// TIA Portal project "TrainingModules2" (V15.1)

(* hardware
DEVICE "S71500/ET200MP station_1"  S7-1500 station
   slot 0: "Rail_0"  Rack  6ES7 590-1***0-0AA0
   slot 1: "PLC_1"  CPU 1516-3 PN/DP  6ES7 516-3AN01-0AB0  V2.6
      slot 3: "CPU display_1"  6ES7591-1BA00-0AA0
*)

// ===== PLC "PLC_1"  CPU 1516-3 PN/DP =====

VAR_GLOBAL   // PLC tag table "Control Panel"
   "Auto Mode" AT %I0.0 : Bool;   // Automaitc Mode Switch
   "Auto Mode Start PB" AT %I0.1 : Bool;   // Auto Mode Start Push Button
   "Auto Mode Stop PB" AT %I0.2 : Bool;   // Auto Mode Stop Push Button
   "Manual Mode" AT %I0.3 : Bool;   // Manual Mode Switch
   "Reset Counter" AT %I0.4 : Bool;   // Reset Part Counter
   "EStop" AT %I0.5 : Bool;   // Emergency Stop
   "Start Light" AT %Q0.0 : Bool;   // Start Push Button Light
   "Stop Light" AT %Q0.1 : Bool;   // Stop Push Button Light
   "Reset Light" AT %Q0.2 : Bool;   // Reset Push Button Light
   "Part Entry Counter" AT %QD100 : DInt;   // Part Entry Counter
   "Garbage" AT %M10.0 : Bool;   // Storage for Last Cycle, Not Used
   "Garbage2" AT %M10.1 : Bool;   // Storage for Last Cycle, Not Used
END_VAR

VAR_GLOBAL   // PLC tag table "Conveyor"
   "Tall Sensor" AT %I0.6 : Bool;   // Second Level Height Sensor
   "Short Sensor" AT %I0.7 : Bool;   // First Level Height Sensor
   "Conveyor_Loader_Entry" AT %I1.2 : Bool;   // Entering the Main Conveyor
   "Conveyor_Left_Entry" AT %I1.3 : Bool;   // Left Conveyor Entry Sensor
   "Conveyor_Right_Entry" AT %I1.4 : Bool;   // Right Conveyor Entry Sensor
   "Conveyor_Turntable_Entry" AT %I1.5 : Bool;   // Entering the Turntable
   "Feeder Conveyor" AT %Q0.3 : Bool;   // Feeder Conveyor Actuator
   "Entry Conveyor" AT %Q0.4 : Bool;   // Entry Conveyor Actuator
   "Left Conveyor" AT %Q1.0 : Bool;   // Left Conveyor Actuator
   "Right Conveyor" AT %Q1.1 : Bool;   // Right Conveyor Actuator
   "Green Indicator" AT %Q1.2 : Bool;   // Green Light Indicator
   "Yellow Indicator" AT %Q1.3 : Bool;   // Yellow Light Indicator
   "Red Indicator" AT %Q1.4 : Bool;   // Red Light Indicator
   "Emitter" AT %Q1.5 : Bool;   // Send Parts
   "Remover Left" AT %Q1.6 : Bool;   // Remove Parts Left Side
   "Remover Right" AT %Q1.7 : Bool;   // Remove Parts Right SIde
END_VAR

VAR_GLOBAL   // PLC tag table "Turntable"
   "TT_Front" AT %I1.0 : Bool;   // Turn Table Entry Sensor
   "TT_Back" AT %I1.1 : Bool;   // Turn Table Exit Sensor
   "Home" AT %I1.6 : Bool;   // Turn Table Homed
   "Rotated" AT %I1.7 : Bool;   // Turn Table Rotated
   "Load (Right)" AT %Q0.5 : Bool;   // Load Right Conveyor (TT)
   "Unload (Left)" AT %Q0.6 : Bool;   // Load Left Conveyor (TT)
   "Turn CC" AT %Q0.7 : Bool;   // Turn Table Rotate Counter CLockwise
END_VAR

VAR_GLOBAL   // PLC tag table "Part Buffer"
   "Part_Space_5" AT %MW0 : Int;   // Part Buffer 5
   "Part_Space_4" AT %MW2 : Int;   // Part Buffer 4
   "Part_Space_3" AT %MW4 : Int;   // Part Buffer 3
   "Part_Space_2" AT %MW6 : Int;   // Part Buffer 2
   "Part_Space_1" AT %MW8 : Int;   // Part Buffer 1
END_VAR

DATA_BLOCK "Data_Organization"   // DB1
{ S7_Optimized_Access := 'TRUE' }
VERSION : 0.1
// stored: InstanceOfName Controller
"Controller"
BEGIN
END_DATA_BLOCK

FUNCTION_BLOCK "Controller"   // FB1, LAD
{ S7_Optimized_Access := 'TRUE' }
VERSION : 0.1
   VAR
      "Conveyor Logic_Feeder" : "Conveyor Logic";
      "Turntable Logic" : "Turntable Logic";
      "Conveyor Logic_Entry" : "Conveyor Logic";
      "Conveyor Logic_Left" : "Conveyor Logic";
      "Conveyor Logic_Right" : "Conveyor Logic";
   END_VAR
   VAR_TEMP   // added for the SCL form of the ladder/FBD networks
      _w1 : Bool;
   END_VAR
BEGIN

REGION Network 1: Call the Send and Receive function
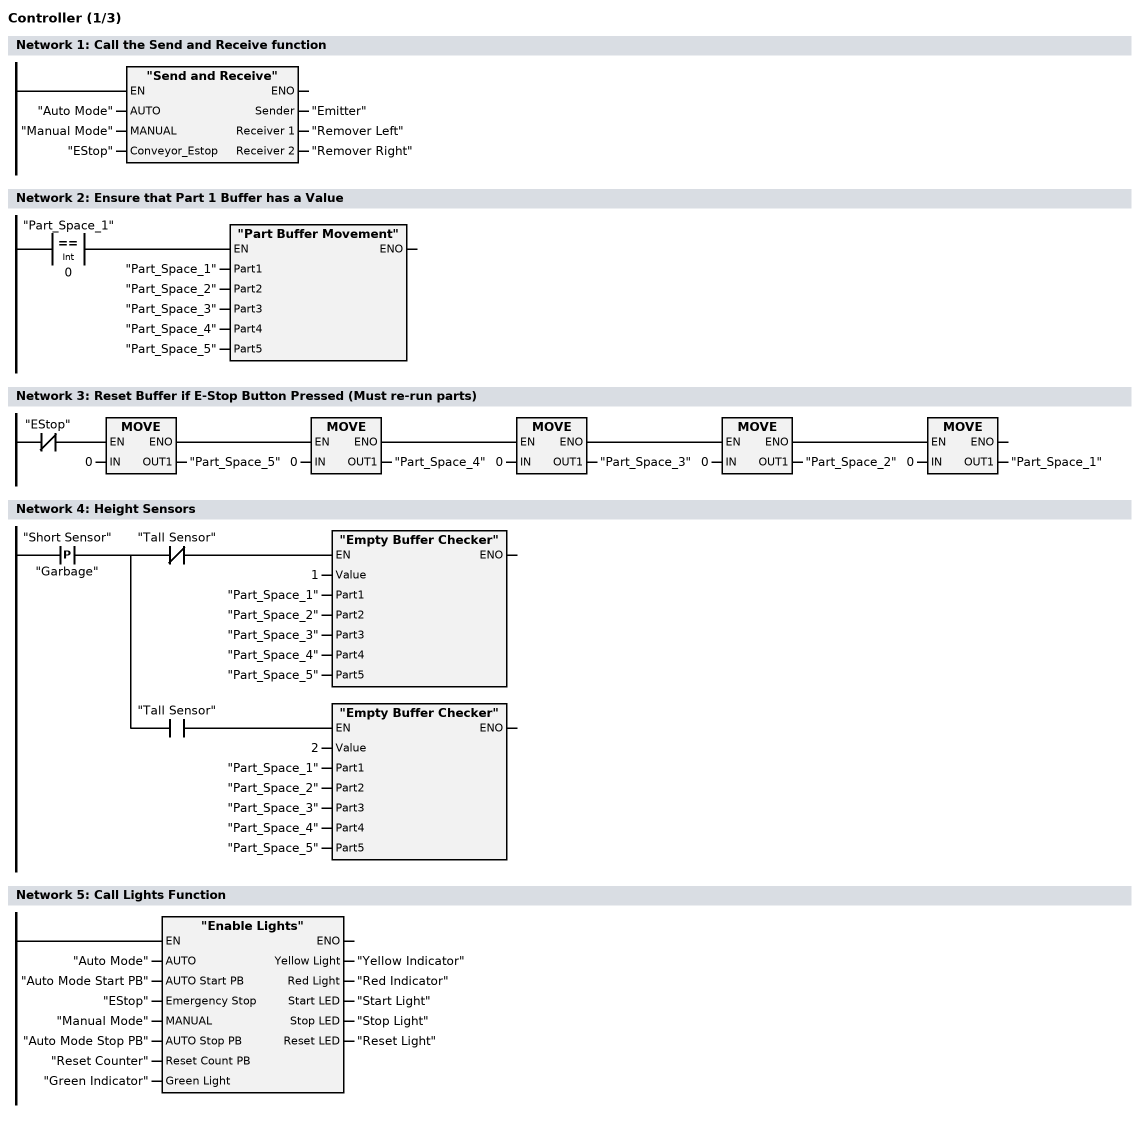
   RUNG wire#powerrail
      "Send and Receive"(AUTO := "Auto Mode", MANUAL := "Manual Mode", Conveyor_Estop := "EStop", Sender => "Emitter", "Receiver 1" => "Remover Left", "Receiver 2" => "Remover Right")
   END_RUNG
   // the same network as SCL:
   "Send and Receive"(AUTO := "Auto Mode",
                      MANUAL := "Manual Mode",
                      Conveyor_Estop := "EStop",
                      Sender => "Emitter",
                      "Receiver 1" => "Remover Left",
                      "Receiver 2" => "Remover Right");
END_REGION

REGION Network 2: Ensure that Part 1 Buffer has a Value
   RUNG wire#powerrail
      { S7_Templates := "SrcType := Int" } EQ_Contact(in1 := "Part_Space_1", in2 := 0)
      "Part Buffer Movement"(Part1 := "Part_Space_1", Part2 := "Part_Space_2", Part3 := "Part_Space_3", Part4 := "Part_Space_4", Part5 := "Part_Space_5")
   END_RUNG
   // the same network as SCL:
   IF "Part_Space_1" = 0 THEN
       "Part Buffer Movement"(Part1 := "Part_Space_1",
                              Part2 := "Part_Space_2",
                              Part3 := "Part_Space_3",
                              Part4 := "Part_Space_4",
                              Part5 := "Part_Space_5");
   END_IF;
END_REGION

REGION Network 3: Reset Buffer if E-Stop Button Pressed (Must re-run parts)
   RUNG wire#powerrail
      I_Contact( "EStop" )
      Move(in := 0, out1 => "Part_Space_5")
      Move(in := 0, out1 => "Part_Space_4")
      Move(in := 0, out1 => "Part_Space_3")
      Move(in := 0, out1 => "Part_Space_2")
      Move(in := 0, out1 => "Part_Space_1")
   END_RUNG
   // the same network as SCL:
   IF NOT "EStop" THEN
       "Part_Space_5" := 0;
       "Part_Space_4" := 0;
       "Part_Space_3" := 0;
       "Part_Space_2" := 0;
       "Part_Space_1" := 0;
   END_IF;
END_REGION

REGION Network 4: Height Sensors
   RUNG wire#powerrail
      P_Contact(operand := "Short Sensor", bit := "Garbage")
      wire#w1
      I_Contact( "Tall Sensor" )
      "Empty Buffer Checker"(Value := 1, Part1 := "Part_Space_1", Part2 := "Part_Space_2", Part3 := "Part_Space_3", Part4 := "Part_Space_4", Part5 := "Part_Space_5")
   END_RUNG
   RUNG wire#w1
      Contact( "Tall Sensor" )
      "Empty Buffer Checker"(Value := 2, Part1 := "Part_Space_1", Part2 := "Part_Space_2", Part3 := "Part_Space_3", Part4 := "Part_Space_4", Part5 := "Part_Space_5")
   END_RUNG
   // the same network as SCL:
   #_w1 := "Short Sensor" AND NOT "Garbage";   // rising edge of "Short Sensor"
   "Garbage" := "Short Sensor";
   IF #_w1 AND NOT "Tall Sensor" THEN
       "Empty Buffer Checker"(Value := 1,
                              Part1 := "Part_Space_1",
                              Part2 := "Part_Space_2",
                              Part3 := "Part_Space_3",
                              Part4 := "Part_Space_4",
                              Part5 := "Part_Space_5");
   END_IF;
   IF #_w1 AND "Tall Sensor" THEN
       "Empty Buffer Checker"(Value := 2,
                              Part1 := "Part_Space_1",
                              Part2 := "Part_Space_2",
                              Part3 := "Part_Space_3",
                              Part4 := "Part_Space_4",
                              Part5 := "Part_Space_5");
   END_IF;
END_REGION

REGION Network 5: Call Lights Function
   RUNG wire#powerrail
      "Enable Lights"(AUTO := "Auto Mode", "AUTO Start PB" := "Auto Mode Start PB", "Emergency Stop" := "EStop", MANUAL := "Manual Mode", "AUTO Stop PB" := "Auto Mode Stop PB", "Reset Count PB" := "Reset Counter", "Green Light" := "Green Indicator", "Yellow Light" => "Yellow Indicator", "Red Light" => "Red Indicator", "Start LED" => "Start Light", "Stop LED" => "Stop Light", "Reset LED" => "Reset Light")
   END_RUNG
   // the same network as SCL:
   "Enable Lights"(AUTO := "Auto Mode",
                   "AUTO Start PB" := "Auto Mode Start PB",
                   "Emergency Stop" := "EStop",
                   MANUAL := "Manual Mode",
                   "AUTO Stop PB" := "Auto Mode Stop PB",
                   "Reset Count PB" := "Reset Counter",
                   "Green Light" := "Green Indicator",
                   "Yellow Light" => "Yellow Indicator",
                   "Red Light" => "Red Indicator",
                   "Start LED" => "Start Light",
                   "Stop LED" => "Stop Light",
                   "Reset LED" => "Reset Light");
END_REGION

REGION Network 6: Call Feeder Conveyor Logic
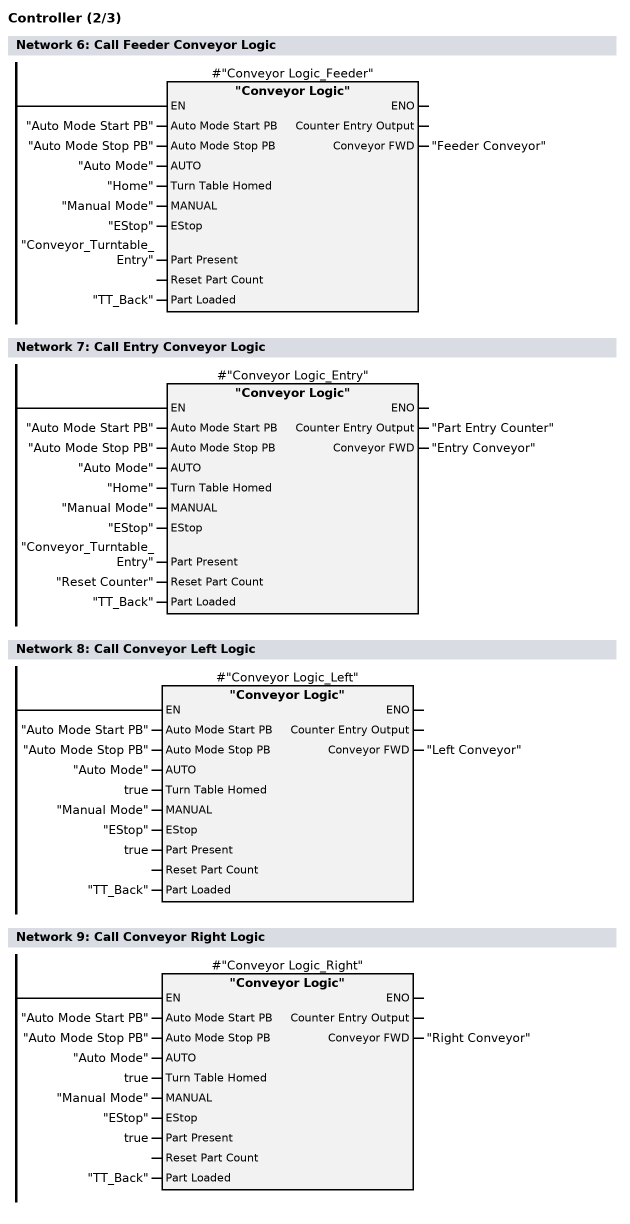
   RUNG wire#powerrail
      #"Conveyor Logic_Feeder"("Auto Mode Start PB" := "Auto Mode Start PB", "Auto Mode Stop PB" := "Auto Mode Stop PB", AUTO := "Auto Mode", "Turn Table Homed" := "Home", MANUAL := "Manual Mode", EStop := "EStop", "Part Present" := "Conveyor_Turntable_Entry", "Reset Part Count" :=, "Part Loaded" := "TT_Back", "Counter Entry Output" =>, "Conveyor FWD" => "Feeder Conveyor")
   END_RUNG
   // the same network as SCL:
   #"Conveyor Logic_Feeder"("Auto Mode Start PB" := "Auto Mode Start PB",   // "Conveyor Logic"
                           "Auto Mode Stop PB" := "Auto Mode Stop PB",
                           AUTO := "Auto Mode",
                           "Turn Table Homed" := "Home",
                           MANUAL := "Manual Mode",
                           EStop := "EStop",
                           "Part Present" := "Conveyor_Turntable_Entry",
                           "Part Loaded" := "TT_Back",
                           "Conveyor FWD" => "Feeder Conveyor");
END_REGION

REGION Network 7: Call Entry Conveyor Logic
   RUNG wire#powerrail
      #"Conveyor Logic_Entry"("Auto Mode Start PB" := "Auto Mode Start PB", "Auto Mode Stop PB" := "Auto Mode Stop PB", AUTO := "Auto Mode", "Turn Table Homed" := "Home", MANUAL := "Manual Mode", EStop := "EStop", "Part Present" := "Conveyor_Turntable_Entry", "Reset Part Count" := "Reset Counter", "Part Loaded" := "TT_Back", "Counter Entry Output" => "Part Entry Counter", "Conveyor FWD" => "Entry Conveyor")
   END_RUNG
   // the same network as SCL:
   #"Conveyor Logic_Entry"("Auto Mode Start PB" := "Auto Mode Start PB",   // "Conveyor Logic"
                           "Auto Mode Stop PB" := "Auto Mode Stop PB",
                           AUTO := "Auto Mode",
                           "Turn Table Homed" := "Home",
                           MANUAL := "Manual Mode",
                           EStop := "EStop",
                           "Part Present" := "Conveyor_Turntable_Entry",
                           "Reset Part Count" := "Reset Counter",
                           "Part Loaded" := "TT_Back",
                           "Counter Entry Output" => "Part Entry Counter",
                           "Conveyor FWD" => "Entry Conveyor");
END_REGION

REGION Network 8: Call Conveyor Left Logic
   RUNG wire#powerrail
      #"Conveyor Logic_Left"("Auto Mode Start PB" := "Auto Mode Start PB", "Auto Mode Stop PB" := "Auto Mode Stop PB", AUTO := "Auto Mode", "Turn Table Homed" := true, MANUAL := "Manual Mode", EStop := "EStop", "Part Present" := true, "Reset Part Count" :=, "Part Loaded" := "TT_Back", "Counter Entry Output" =>, "Conveyor FWD" => "Left Conveyor")
   END_RUNG
   // the same network as SCL:
   #"Conveyor Logic_Left"("Auto Mode Start PB" := "Auto Mode Start PB",   // "Conveyor Logic"
                          "Auto Mode Stop PB" := "Auto Mode Stop PB",
                          AUTO := "Auto Mode",
                          "Turn Table Homed" := true,
                          MANUAL := "Manual Mode",
                          EStop := "EStop",
                          "Part Present" := true,
                          "Part Loaded" := "TT_Back",
                          "Conveyor FWD" => "Left Conveyor");
END_REGION

REGION Network 9: Call Conveyor Right Logic
   RUNG wire#powerrail
      #"Conveyor Logic_Right"("Auto Mode Start PB" := "Auto Mode Start PB", "Auto Mode Stop PB" := "Auto Mode Stop PB", AUTO := "Auto Mode", "Turn Table Homed" := true, MANUAL := "Manual Mode", EStop := "EStop", "Part Present" := true, "Reset Part Count" :=, "Part Loaded" := "TT_Back", "Counter Entry Output" =>, "Conveyor FWD" => "Right Conveyor")
   END_RUNG
   // the same network as SCL:
   #"Conveyor Logic_Right"("Auto Mode Start PB" := "Auto Mode Start PB",   // "Conveyor Logic"
                           "Auto Mode Stop PB" := "Auto Mode Stop PB",
                           AUTO := "Auto Mode",
                           "Turn Table Homed" := true,
                           MANUAL := "Manual Mode",
                           EStop := "EStop",
                           "Part Present" := true,
                           "Part Loaded" := "TT_Back",
                           "Conveyor FWD" => "Right Conveyor");
END_REGION

REGION Network 10: Call Turntable Logic
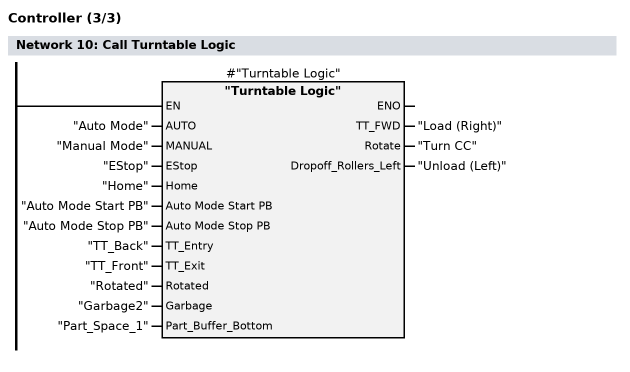
   RUNG wire#powerrail
      #"Turntable Logic"(AUTO := "Auto Mode", MANUAL := "Manual Mode", EStop := "EStop", Home := "Home", "Auto Mode Start PB" := "Auto Mode Start PB", "Auto Mode Stop PB" := "Auto Mode Stop PB", TT_Entry := "TT_Back", TT_Exit := "TT_Front", Rotated := "Rotated", Garbage := "Garbage2", Part_Buffer_Bottom := "Part_Space_1", TT_FWD => "Load (Right)", Rotate => "Turn CC", Dropoff_Rollers_Left => "Unload (Left)")
   END_RUNG
   // the same network as SCL:
   #"Turntable Logic"(AUTO := "Auto Mode",   // "Turntable Logic"
                      MANUAL := "Manual Mode",
                      EStop := "EStop",
                      Home := "Home",
                      "Auto Mode Start PB" := "Auto Mode Start PB",
                      "Auto Mode Stop PB" := "Auto Mode Stop PB",
                      TT_Entry := "TT_Back",
                      TT_Exit := "TT_Front",
                      Rotated := "Rotated",
                      Garbage := "Garbage2",
                      Part_Buffer_Bottom := "Part_Space_1",
                      TT_FWD => "Load (Right)",
                      Rotate => "Turn CC",
                      Dropoff_Rollers_Left => "Unload (Left)");
END_REGION
END_FUNCTION_BLOCK

FUNCTION_BLOCK "Turntable Logic"   // FB2, LAD
{ S7_Optimized_Access := 'TRUE' }
VERSION : 0.1
   VAR_INPUT
      AUTO : Bool;
      MANUAL : Bool;
      EStop : Bool;
      Home : Bool;
      "Auto Mode Start PB" : Bool;
      "Auto Mode Stop PB" : Bool;
      TT_Entry : Bool;
      TT_Exit : Bool;
      Rotated : Bool;
   END_VAR
   VAR_OUTPUT
      TT_FWD : Bool;
      Rotate : Bool;
      Dropoff_Rollers_Left : Bool;
   END_VAR
   VAR_IN_OUT
      Garbage : Bool;
      Part_Buffer_Bottom : Int;
   END_VAR
   VAR
      "Elapsed TIme" : DInt;
      "Auto Stopped" : Bool;
      "Turn Table Timers" : TP_TIME;
      "Load Table" : Bool;
      Dropoff_Rollers_Right : Bool;
      "Rotation Ready" : Bool;
   END_VAR
   VAR_TEMP   // added for the SCL form of the ladder/FBD networks
      _w1 : Bool;
   END_VAR
BEGIN

REGION Network 1: Enable FWD Loading Rollers on Turn Tables
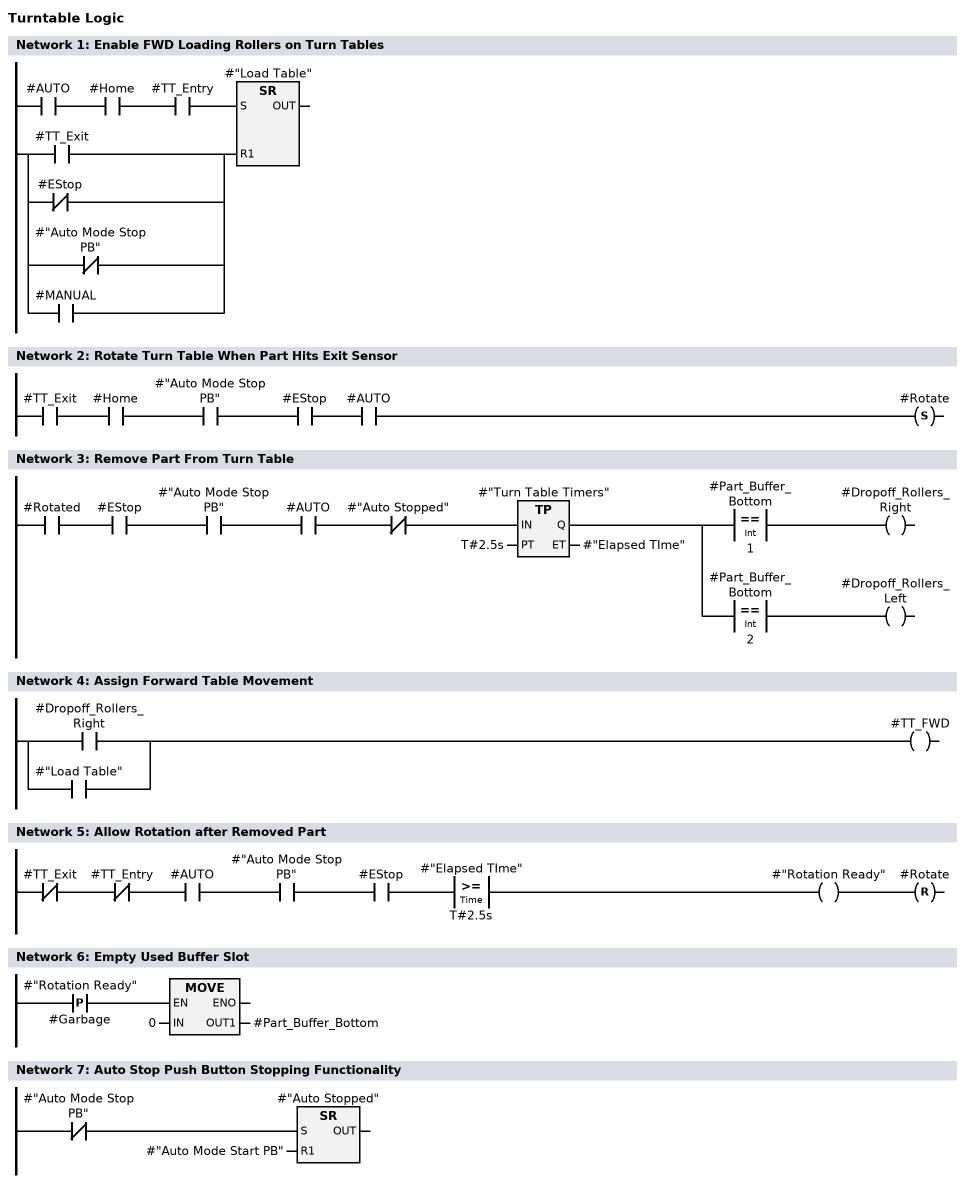
   RUNG wire#powerrail
      Contact( #AUTO )
      Contact( #Home )
      Contact( #TT_Entry )
      S_SR(operand := #"Load Table", r1 := wire#w1)
   END_RUNG
   RUNG wire#powerrail
      Contact( #TT_Exit )
   END_RUNG wire#w1
   RUNG wire#powerrail
      I_Contact( #EStop )
   END_RUNG wire#w1
   RUNG wire#powerrail
      I_Contact( #"Auto Mode Stop PB" )
   END_RUNG wire#w1
   RUNG wire#powerrail
      Contact( #MANUAL )
   END_RUNG wire#w1
   // the same network as SCL:
   IF #AUTO AND #Home AND #TT_Entry THEN
       #"Load Table" := TRUE;   // SR flip-flop
   END_IF;
   IF #TT_Exit OR NOT #EStop OR NOT #"Auto Mode Stop PB" OR #MANUAL THEN #"Load Table" := FALSE; END_IF;
END_REGION

REGION Network 2: Rotate Turn Table When Part Hits Exit Sensor
   RUNG wire#powerrail
      Contact( #TT_Exit )
      Contact( #Home )
      Contact( #"Auto Mode Stop PB" )
      Contact( #EStop )
      Contact( #AUTO )
      S_Coil( #Rotate )
   END_RUNG
   // the same network as SCL:
   IF #TT_Exit AND #Home AND #"Auto Mode Stop PB" AND #EStop AND #AUTO THEN #Rotate := TRUE; END_IF;
END_REGION

REGION Network 3: Remove Part From Turn Table
   #"Turn Table Timers"(IN := #Rotated AND #EStop AND #"Auto Mode Stop PB" AND #AUTO AND NOT #"Auto Stopped",   // TP
                        PT := T#2.5s,
                        ET => #"Elapsed TIme");
   #Dropoff_Rollers_Right := #"Turn Table Timers".Q AND (#Part_Buffer_Bottom = 1);
   #Dropoff_Rollers_Left := #"Turn Table Timers".Q AND (#Part_Buffer_Bottom = 2);
END_REGION

REGION Network 4: Assign Forward Table Movement
   RUNG wire#powerrail
      Contact( #Dropoff_Rollers_Right )
      wire#w1
      Coil( #TT_FWD )
   END_RUNG
   RUNG wire#powerrail
      Contact( #"Load Table" )
   END_RUNG wire#w1
   // the same network as SCL:
   #TT_FWD := #Dropoff_Rollers_Right OR #"Load Table";
END_REGION

REGION Network 5: Allow Rotation after Removed Part
   RUNG wire#powerrail
      I_Contact( #TT_Exit )
      I_Contact( #TT_Entry )
      Contact( #AUTO )
      Contact( #"Auto Mode Stop PB" )
      Contact( #EStop )
      { S7_Templates := "SrcType := Time" } GE_Contact(in1 := #"Elapsed TIme", in2 := T#2.5s)
      Coil( #"Rotation Ready" )
      R_Coil( #Rotate )
   END_RUNG
   // the same network as SCL:
   #"Rotation Ready" := NOT #TT_Exit AND NOT #TT_Entry AND #AUTO AND #"Auto Mode Stop PB" AND #EStop AND (#"Elapsed TIme" >= T#2.5s);
   IF #"Rotation Ready" THEN #Rotate := FALSE; END_IF;
END_REGION

REGION Network 6: Empty Used Buffer Slot
   RUNG wire#powerrail
      P_Contact(operand := #"Rotation Ready", bit := #Garbage)
      Move(in := 0, out1 => #Part_Buffer_Bottom)
   END_RUNG
   // the same network as SCL:
   #_w1 := #"Rotation Ready" AND NOT #Garbage;   // rising edge of #"Rotation Ready"
   #Garbage := #"Rotation Ready";
   IF #_w1 THEN #Part_Buffer_Bottom := 0; END_IF;
END_REGION

REGION Network 7: Auto Stop Push Button Stopping Functionality
   RUNG wire#powerrail
      I_Contact( #"Auto Mode Stop PB" )
      S_SR(operand := #"Auto Stopped", r1 := #"Auto Mode Start PB")
   END_RUNG
   // the same network as SCL:
   IF NOT #"Auto Mode Stop PB" THEN
       #"Auto Stopped" := TRUE;   // SR flip-flop
   END_IF;
   IF #"Auto Mode Start PB" THEN #"Auto Stopped" := FALSE; END_IF;
END_REGION
END_FUNCTION_BLOCK

FUNCTION_BLOCK "Conveyor Logic"   // FB3, LAD
{ S7_Optimized_Access := 'TRUE' }
VERSION : 0.1
   VAR_INPUT
      "Auto Mode Start PB" : Bool;
      "Auto Mode Stop PB" : Bool;
      AUTO : Bool;
      "Turn Table Homed" : Bool;
      MANUAL : Bool;
      EStop : Bool;
      "Part Present" : Bool;
      "Reset Part Count" : Bool;
      "Part Loaded" : Bool;
   END_VAR
   VAR_OUTPUT
      "Counter Entry Output" : Int;
      "Conveyor FWD" : Bool;
   END_VAR
   VAR
      "Conveyor Started" : Bool;
   END_VAR
   VAR RETAIN
      "Part Entry Counter" : CTU_INT;
   END_VAR
BEGIN

REGION Network 1: Conveyor Auto Mode
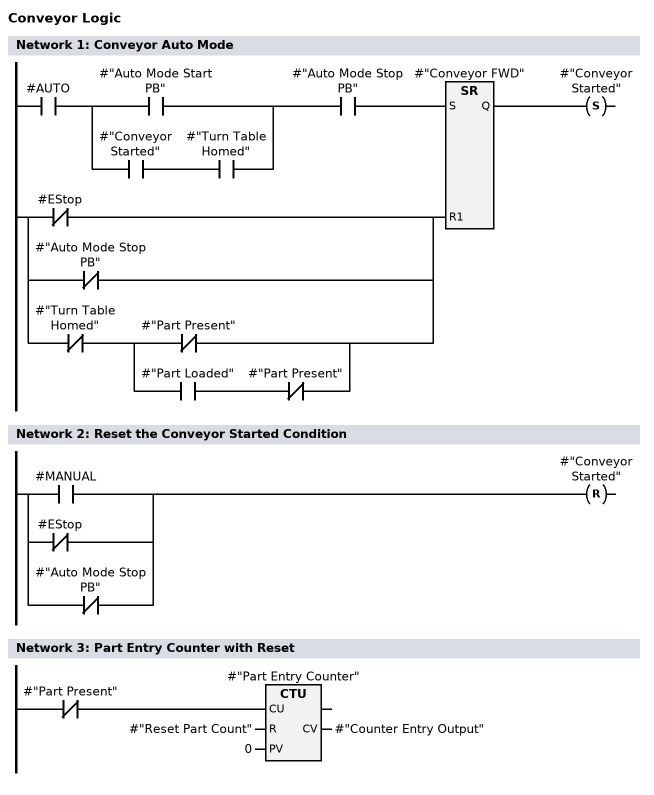
   RUNG wire#powerrail
      Contact( #AUTO )
      wire#w1
      Contact( #"Auto Mode Start PB" )
      wire#w2
      Contact( #"Auto Mode Stop PB" )
      S_SR(operand := #"Conveyor FWD", r1 := wire#w4)
      S_Coil( #"Conveyor Started" )
   END_RUNG
   RUNG wire#w1
      Contact( #"Conveyor Started" )
      Contact( #"Turn Table Homed" )
   END_RUNG wire#w2
   RUNG wire#powerrail
      I_Contact( #EStop )
   END_RUNG wire#w4
   RUNG wire#powerrail
      I_Contact( #"Auto Mode Stop PB" )
   END_RUNG wire#w4
   RUNG wire#powerrail
      I_Contact( #"Turn Table Homed" )
      wire#w3
      I_Contact( #"Part Present" )
   END_RUNG wire#w4
   RUNG wire#w3
      Contact( #"Part Loaded" )
      I_Contact( #"Part Present" )
   END_RUNG wire#w4
   // the same network as SCL:
   IF #AUTO AND (#"Auto Mode Start PB" OR (#"Conveyor Started" AND #"Turn Table Homed")) AND #"Auto Mode Stop PB" THEN
       #"Conveyor FWD" := TRUE;   // SR flip-flop
   END_IF;
   IF NOT #EStop OR NOT #"Auto Mode Stop PB" OR (NOT #"Turn Table Homed" AND (NOT #"Part Present" OR (#"Part Loaded" AND NOT #"Part Present"))) THEN
       #"Conveyor FWD" := FALSE;
   END_IF;
   IF #"Conveyor FWD" THEN #"Conveyor Started" := TRUE; END_IF;
END_REGION

REGION Network 2: Reset the Conveyor Started Condition
   RUNG wire#powerrail
      Contact( #MANUAL )
      wire#w1
      R_Coil( #"Conveyor Started" )
   END_RUNG
   RUNG wire#powerrail
      I_Contact( #EStop )
   END_RUNG wire#w1
   RUNG wire#powerrail
      I_Contact( #"Auto Mode Stop PB" )
   END_RUNG wire#w1
   // the same network as SCL:
   IF #MANUAL OR NOT #EStop OR NOT #"Auto Mode Stop PB" THEN #"Conveyor Started" := FALSE; END_IF;
END_REGION

REGION Network 3: Part Entry Counter with Reset
   #"Part Entry Counter"(CU := NOT #"Part Present",   // CTU
                         R := #"Reset Part Count",
                         PV := 0,
                         CV => #"Counter Entry Output");
END_REGION
END_FUNCTION_BLOCK

FUNCTION "Send and Receive" : Void   // FC1, LAD
{ S7_Optimized_Access := 'TRUE' }
VERSION : 0.1
   VAR_INPUT
      AUTO : Bool;
      MANUAL : Bool;
      Conveyor_Estop : Bool;
   END_VAR
   VAR_OUTPUT
      Sender : Bool;
      "Receiver 1" : Bool;
      "Receiver 2" : Bool;
   END_VAR
BEGIN

REGION Network 1: Send and Receive Parts in Auto Mode
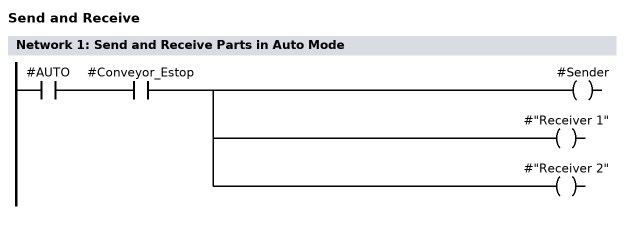
   RUNG wire#powerrail
      Contact( #AUTO )
      Contact( #Conveyor_Estop )
      wire#w1
      Coil( #Sender )
   END_RUNG
   RUNG wire#w1
      Coil( #"Receiver 1" )
   END_RUNG
   RUNG wire#w1
      Coil( #"Receiver 2" )
   END_RUNG
   // the same network as SCL:
   #Sender := #AUTO AND #Conveyor_Estop;
   #"Receiver 1" := #Sender;
   #"Receiver 2" := #Sender;
END_REGION
END_FUNCTION

FUNCTION "Part Buffer Movement" : Void   // FC2, LAD
{ S7_Optimized_Access := 'TRUE' }
VERSION : 0.1
   VAR_IN_OUT
      Part1 : Int;
      Part2 : Int;
      Part3 : Int;
      Part4 : Int;
      Part5 : Int;
   END_VAR
   VAR_TEMP
      Part4Temp : Int;
      Part3Temp : Int;
      Part2Temp : Int;
      Part1Temp : Int;
   END_VAR
BEGIN

REGION Network 1: Shift Part Buffer
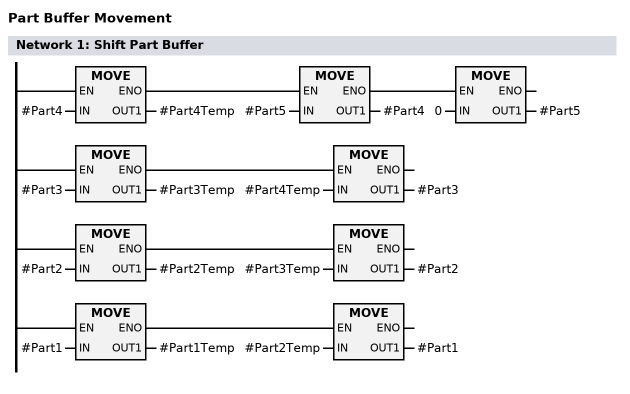
   RUNG wire#powerrail
      Move(in := #Part4, out1 => #Part4Temp)
      Move(in := #Part5, out1 => #Part4)
      Move(in := 0, out1 => #Part5)
   END_RUNG
   RUNG wire#powerrail
      Move(in := #Part3, out1 => #Part3Temp)
      Move(in := #Part4Temp, out1 => #Part3)
   END_RUNG
   RUNG wire#powerrail
      Move(in := #Part2, out1 => #Part2Temp)
      Move(in := #Part3Temp, out1 => #Part2)
   END_RUNG
   RUNG wire#powerrail
      Move(in := #Part1, out1 => #Part1Temp)
      Move(in := #Part2Temp, out1 => #Part1)
   END_RUNG
   // the same network as SCL:
   #Part4Temp := #Part4;
   #Part4 := #Part5;
   #Part5 := 0;
   #Part3Temp := #Part3;
   #Part3 := #Part4Temp;
   #Part2Temp := #Part2;
   #Part2 := #Part3Temp;
   #Part1Temp := #Part1;
   #Part1 := #Part2Temp;
END_REGION
END_FUNCTION

FUNCTION "Enable Lights" : Void   // FC3, LAD
{ S7_Optimized_Access := 'TRUE' }
VERSION : 0.1
   VAR_INPUT
      AUTO : Bool;
      "AUTO Start PB" : Bool;
      "Emergency Stop" : Bool;
      MANUAL : Bool;
      "AUTO Stop PB" : Bool;
      "Reset Count PB" : Bool;
   END_VAR
   VAR_OUTPUT
      "Yellow Light" : Bool;
      "Red Light" : Bool;
      "Start LED" : Bool;
      "Stop LED" : Bool;
      "Reset LED" : Bool;
   END_VAR
   VAR_IN_OUT
      "Green Light" : Bool;
   END_VAR
BEGIN

REGION Network 1: Enable Green Light (Auto)
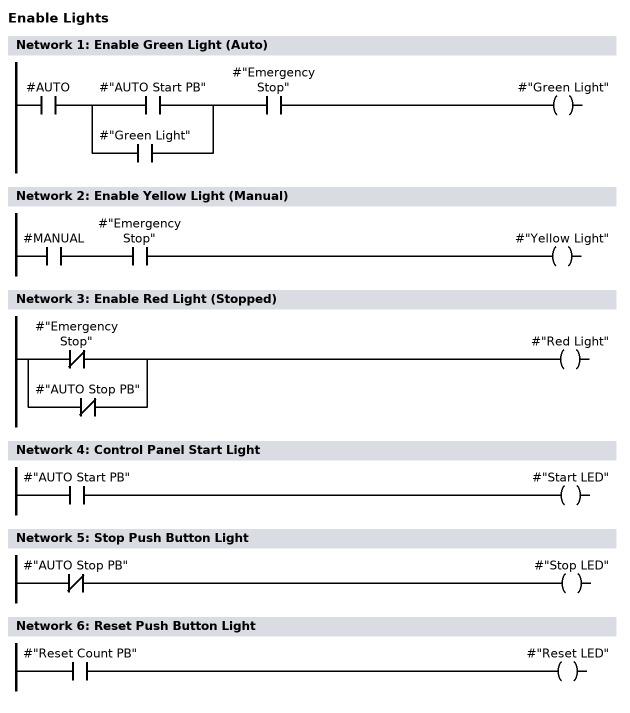
   RUNG wire#powerrail
      Contact( #AUTO )
      wire#w1
      Contact( #"AUTO Start PB" )
      wire#w2
      Contact( #"Emergency Stop" )
      Coil( #"Green Light" )
   END_RUNG
   RUNG wire#w1
      Contact( #"Green Light" )
   END_RUNG wire#w2
   // the same network as SCL:
   #"Green Light" := #AUTO AND (#"AUTO Start PB" OR #"Green Light") AND #"Emergency Stop";
END_REGION

REGION Network 2: Enable Yellow Light (Manual)
   RUNG wire#powerrail
      Contact( #MANUAL )
      Contact( #"Emergency Stop" )
      Coil( #"Yellow Light" )
   END_RUNG
   // the same network as SCL:
   #"Yellow Light" := #MANUAL AND #"Emergency Stop";
END_REGION

REGION Network 3: Enable Red Light (Stopped)
   RUNG wire#powerrail
      I_Contact( #"Emergency Stop" )
      wire#w1
      Coil( #"Red Light" )
   END_RUNG
   RUNG wire#powerrail
      I_Contact( #"AUTO Stop PB" )
   END_RUNG wire#w1
   // the same network as SCL:
   #"Red Light" := NOT #"Emergency Stop" OR NOT #"AUTO Stop PB";
END_REGION

REGION Network 4: Control Panel Start Light
   RUNG wire#powerrail
      Contact( #"AUTO Start PB" )
      Coil( #"Start LED" )
   END_RUNG
   // the same network as SCL:
   #"Start LED" := #"AUTO Start PB";
END_REGION

REGION Network 5: Stop Push Button Light
   RUNG wire#powerrail
      I_Contact( #"AUTO Stop PB" )
      Coil( #"Stop LED" )
   END_RUNG
   // the same network as SCL:
   #"Stop LED" := NOT #"AUTO Stop PB";
END_REGION

REGION Network 6: Reset Push Button Light
   RUNG wire#powerrail
      Contact( #"Reset Count PB" )
      Coil( #"Reset LED" )
   END_RUNG
   // the same network as SCL:
   #"Reset LED" := #"Reset Count PB";
END_REGION
END_FUNCTION

FUNCTION "Empty Buffer Checker" : Void   // FC4, LAD
{ S7_Optimized_Access := 'TRUE' }
VERSION : 0.1
   VAR_INPUT
      Value : Int;
   END_VAR
   VAR_IN_OUT
      Part1 : Int;
      Part2 : Int;
      Part3 : Int;
      Part4 : Int;
      Part5 : Int;
   END_VAR
BEGIN

REGION Network 1: Empty Buffer Checker
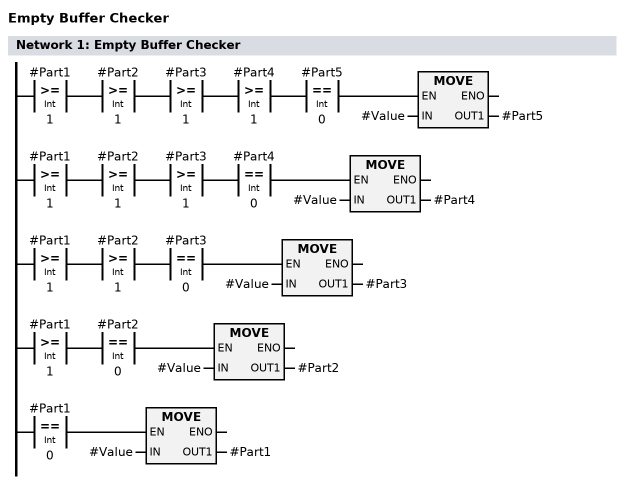
   RUNG wire#powerrail
      { S7_Templates := "SrcType := Int" } GE_Contact(in1 := #Part1, in2 := 1)
      { S7_Templates := "SrcType := Int" } GE_Contact(in1 := #Part2, in2 := 1)
      { S7_Templates := "SrcType := Int" } GE_Contact(in1 := #Part3, in2 := 1)
      { S7_Templates := "SrcType := Int" } GE_Contact(in1 := #Part4, in2 := 1)
      { S7_Templates := "SrcType := Int" } EQ_Contact(in1 := #Part5, in2 := 0)
      Move(in := #Value, out1 => #Part5)
   END_RUNG
   RUNG wire#powerrail
      { S7_Templates := "SrcType := Int" } GE_Contact(in1 := #Part1, in2 := 1)
      { S7_Templates := "SrcType := Int" } GE_Contact(in1 := #Part2, in2 := 1)
      { S7_Templates := "SrcType := Int" } GE_Contact(in1 := #Part3, in2 := 1)
      { S7_Templates := "SrcType := Int" } EQ_Contact(in1 := #Part4, in2 := 0)
      Move(in := #Value, out1 => #Part4)
   END_RUNG
   RUNG wire#powerrail
      { S7_Templates := "SrcType := Int" } GE_Contact(in1 := #Part1, in2 := 1)
      { S7_Templates := "SrcType := Int" } GE_Contact(in1 := #Part2, in2 := 1)
      { S7_Templates := "SrcType := Int" } EQ_Contact(in1 := #Part3, in2 := 0)
      Move(in := #Value, out1 => #Part3)
   END_RUNG
   RUNG wire#powerrail
      { S7_Templates := "SrcType := Int" } GE_Contact(in1 := #Part1, in2 := 1)
      { S7_Templates := "SrcType := Int" } EQ_Contact(in1 := #Part2, in2 := 0)
      Move(in := #Value, out1 => #Part2)
   END_RUNG
   RUNG wire#powerrail
      { S7_Templates := "SrcType := Int" } EQ_Contact(in1 := #Part1, in2 := 0)
      Move(in := #Value, out1 => #Part1)
   END_RUNG
   // the same network as SCL:
   IF (#Part1 >= 1) AND (#Part2 >= 1) AND (#Part3 >= 1) AND (#Part4 >= 1) AND (#Part5 = 0) THEN
       #Part5 := #Value;
   END_IF;
   IF (#Part1 >= 1) AND (#Part2 >= 1) AND (#Part3 >= 1) AND (#Part4 = 0) THEN #Part4 := #Value; END_IF;
   IF (#Part1 >= 1) AND (#Part2 >= 1) AND (#Part3 = 0) THEN #Part3 := #Value; END_IF;
   IF (#Part1 >= 1) AND (#Part2 = 0) THEN #Part2 := #Value; END_IF;
   IF #Part1 = 0 THEN #Part1 := #Value; END_IF;
END_REGION
END_FUNCTION

ORGANIZATION_BLOCK "Main"   // OB1, LAD, ProgramCycle
TITLE = "Main Program Sweep (Cycle)"
{ S7_Optimized_Access := 'TRUE' }
VERSION : 0.1
   VAR_INPUT
      Initial_Call : Bool;   // Initial call of this OB
      Remanence : Bool;   // =True, if remanent data are available
   END_VAR
BEGIN

REGION Network 1: Call Line Controller
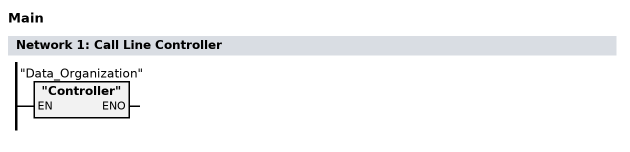
   RUNG wire#powerrail
      "Data_Organization"()
   END_RUNG
   // the same network as SCL:
   "Data_Organization"();   // "Controller"
END_REGION
END_ORGANIZATION_BLOCK